FUNCTION_BLOCK TwoConCtlCentralClient (* Composite Function Block Type *)
  (* Standard: 61499-2 *)
  (* Version 0.2, 2003-12-05, JHC, Rockwell Automation, Renamed from NEWCOMPFB. *)
  (* Version 0.1, 2002-01-08, JHC, Rockwell Automation, Added DLY FB as example. *)
  (* Version 0.0, 2000-05-27, JHC, Rockwell Automation *)
  (* Compiler header: package fb.rt.cs725; *)
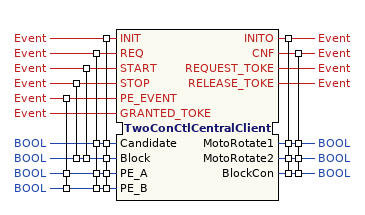
  EVENT_INPUT
    INIT WITH Candidate, Block, PE_A, PE_B; (* Initialization Request *)
    REQ WITH Candidate, PE_A, PE_B; (* Normal Execution Request *)
    START WITH Block;
    STOP WITH Block;
    PE_EVENT WITH PE_A, PE_B;
    GRANTED_TOKE;
  END_EVENT
  EVENT_OUTPUT
    INITO WITH MotoRotate1, MotoRotate2, BlockCon; (* Initialization Confirm *)
    CNF WITH MotoRotate1, MotoRotate2, BlockCon; (* Execution Confirmation *)
    REQUEST_TOKE;
    RELEASE_TOKE;
  END_EVENT
  VAR_INPUT
    Candidate : BOOL;
    Block : BOOL;
    PE_A : BOOL;
    PE_B : BOOL;
  END_VAR
  VAR_OUTPUT
    MotoRotate1 : BOOL;
    MotoRotate2 : BOOL;
    BlockCon : BOOL;
  END_VAR
  FBS
    FC11 : ConveyorCTL(Candidate := 0, Block := 0, PE := 0);
    Conv2Ctl : ConveyorCTLCentralClient;
  END_FBS
  EVENT_CONNECTIONS
    INIT TO FC11.INIT;
    REQ TO FC11.REQ;
    Conv2Ctl.INITO TO INITO;
    Conv2Ctl.CNF TO CNF;
    REQ TO Conv2Ctl.REQ;
    STOP TO Conv2Ctl.CAS_STOP;
    START TO Conv2Ctl.CAS_START;
    Conv2Ctl.STOP TO FC11.CAS_STOP;
    Conv2Ctl.START TO FC11.CAS_START;
    FC11.INITO TO Conv2Ctl.INIT;
    PE_EVENT TO Conv2Ctl.I_PE_EVENT;
    Conv2Ctl.REQUEST_TOKE TO REQUEST_TOKE;
    Conv2Ctl.RELEASE_TOKE TO RELEASE_TOKE;
    GRANTED_TOKE TO Conv2Ctl.GRANTED_TOKE;
  END_CONNECTIONS
  DATA_CONNECTIONS
    Block TO Conv2Ctl.Block;
    Candidate TO Conv2Ctl.Candidate;
    Conv2Ctl.BlockCon TO BlockCon;
    FC11.MotoRotate TO MotoRotate1;
    Conv2Ctl.MotoRotate TO MotoRotate2;
    PE_A TO Conv2Ctl.PE_IN;
    PE_B TO Conv2Ctl.PE_OUT;
  END_CONNECTIONS
END_FUNCTION_BLOCK
